FUNCTION F_ArmsInLoadOrientation : BOOL
VAR_INPUT
END_VAR
VAR
END_VAR

END_FUNCTION

(* stored: Version 1.1.0.1, ProductVersion 3.1.4024.12
   POU F_ArmsInLoadOrientation: Id {da158143-06ca-441d-bcfe-88e196ad8603}, SpecialFunc None *)
